PROGRAM StartStop_Circuit
VAR
	Start: BOOL;
	Stop: BOOL;
	Run_: BOOL;
	
	//Stoppivetoinen versio
	NO_start_button: BOOL;
	NC_Stop_button: BOOL;
END_VAR

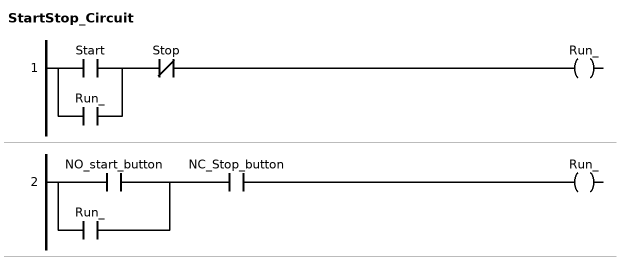
// NETWORK 1
Run_ := (Start OR Run_) AND NOT Stop;

// NETWORK 2
Run_ := (NO_start_button OR Run_) AND NC_Stop_button;

END_PROGRAM

(* stored: Version 1.1.0.1, ProductVersion 3.1.4024.10
   POU StartStop_Circuit: Id {e8d603e0-76da-4b33-a60c-476f61237f8f}, SpecialFunc None *)
